{attribute 'linkalways'} 
{attribute 'no_explicit_call' := 'This FB is a CLASS and must be accessed using methods or properties'}
{attribute 'enable_dynamic_creation'}
FUNCTION_BLOCK _TcVnArray33_UDINT EXTENDS AliasDatatypeBase
VAR
	localData : TcVnArray33_UDINT;
	activeData : REFERENCE TO TcVnArray33_UDINT REF= localData;
	aliasBaseDatatype : _Array0to32OfUDINT;
END_VAR

PROPERTY PUBLIC Address : PVOID
GET
Address := ADR(activeData);
END_GET
END_PROPERTY

METHOD PUBLIC ClearReference
VAR_INPUT
END_VAR
activeData REF= localData;
SetBaseDatatypeReference();
END_METHOD

METHOD PUBLIC Clone : I_Datatype
VAR
    pClone : POINTER TO _TcVnArray33_UDINT;
END_VAR
pClone := __NEW(_TcVnArray33_UDINT);
Clone := pClone^;
END_METHOD

METHOD FB_init : BOOL
VAR_INPUT
	bInitRetains : BOOL; // if TRUE, the retain variables are initialized (warm start / cold start)
	bInCopyCode : BOOL;  // if TRUE, the instance afterwards gets moved into the copy code (online change)
	//InitialValue : TcVnArray33_UDINT; // if possible, not all values can be initialized
END_VAR
//localData := InitialValue; // if possible, not all values can be initialized
SetBaseDatatypeReference();
AddBaseDatatype(aliasBaseDatatype);
END_METHOD

PROPERTY PUBLIC Identifier : T_MAXSTRING
GET
Identifier := 'TcVnArray33_UDINT';
END_GET
END_PROPERTY

METHOD PUBLIC MakeReferenceTo
VAR_INPUT
	ReferenceTarget : REFERENCE TO TcVnArray33_UDINT;
END_VAR
activeData REF= ReferenceTarget;
SetBaseDatatypeReference();
END_METHOD

METHOD PROTECTED SetBaseDatatypeReference
VAR_INPUT
END_VAR
aliasBaseDatatype.MakeReferenceTo(activeData);
END_METHOD

PROPERTY PUBLIC Size : UDINT
GET
Size := SIZEOF(activeData);
END_GET
END_PROPERTY

METHOD TryMakeReferenceTo : BOOL
VAR_INPUT
	Target : I_Datatype;
END_VAR
VAR
	targetAsAlias : I_AliasDatatype;
	pTargetData : POINTER TO TcVnArray33_UDINT;
END_VAR
IF NOT Target.TryResolveAsAliasDatatype(targetAsAlias) THEN
	RETURN;
END_IF

IF targetAsAlias.Identifier <> Identifier THEN
	RETURN;
END_IF

pTargetData := Target.Address;
activeData REF= pTargetData^;
SetBaseDatatypeReference();
TryMakeReferenceTo := TRUE;
END_METHOD

PROPERTY PUBLIC Value : REFERENCE TO TcVnArray33_UDINT
GET
Value REF= activeData;
END_GET
END_PROPERTY

END_FUNCTION_BLOCK

(* stored: Version 1.1.0.1, ProductVersion 3.1.4024.13
   POU _TcVnArray33_UDINT: Id {62f96403-5269-0aab-02c3-1d11c6c243d3}, SpecialFunc None
   Folder Core: Id {c98e78e1-dd26-0595-2eee-89514979cf29}
   Folder Protected: Id {6be008dc-44d4-0fc8-2284-3c36b09efd4d}
   Folder Customize: Id {c9264ef7-d39d-0641-0c3d-9227a8770fbe}
   Folder Constructor: Id {20f6be6a-79ce-01a7-2262-e1f482ffe737}
   Property Address: Id {9ddfdb87-23bc-0ee3-0181-d40dfa9511ea}
   Get Get: Id {ed0ea717-93d1-0860-31a6-84e255c3dc7d}
   Method ClearReference: Id {a7b75c7a-2671-013c-0f27-bf68fc36200c}
   Method Clone: Id {a1afc107-fb9a-0964-3193-8b6bb3d65202}
   Method FB_init: Id {713452c1-41ae-0303-0e96-c36ff8f93984}
   Property Identifier: Id {fa49afe0-fa1c-0bf5-1494-8f747369c27f}
   Get Get: Id {9a18361a-0285-0184-0525-18eb4b511cd8}
   Method MakeReferenceTo: Id {606c2711-a9f6-0854-1ff8-6c300bb7aa22}
   Method SetBaseDatatypeReference: Id {2ebfac0a-8472-0d67-1256-54aaae63467b}
   Property Size: Id {5c65073d-b349-0b93-37b7-0d2206854cd9}
   Get Get: Id {a08c9bab-7ade-051e-09ec-615a5c54c463}
   Method TryMakeReferenceTo: Id {a03d7dc6-5a4d-074e-07eb-bea74ef36f25}
   Property Value: Id {02f120e6-f30b-0c22-1744-5b7eee342036}
   Get Get: Id {658700d0-6e83-063b-1de8-cde1c2dd2d0f} *)
